(* PLC project Generated.project, CODESYS CODESYS V3.5 SP19 Patch 1 *)
(* stored: creationDateTime 2026-09-19T18:18:07.257453, modificationDateTime 2026-09-19T18:18:07.257453 *)

(* ═══════════════════════════════════════════════════════════════ 🧩 ST_fbWinchCmdArbitration_Context — Contexte de gating treuil (partagé M1/M2) ─────────────────────────────────────────────────────────────── 🎯 Rôle : Encapsuler les faits de gating consommés par FB_WinchCommandArbitrationM1/M2 (benne, synchro, blocage both). Structure UNIQUE partagée par les 2 axes, identifiée par l'instance : M1 ignore le chemin benne, M2 le consomme. 📤 Producteur : PRG_04_Treuils_Benne (câblage). 📄 Doc : DOC/AF/AF_Partie-10_Fonction_Winch_v2.1.md 🔌 Action benne : 2 bits BOOL directionnels M2 issus de FB_Bucket. ═══════════════════════════════════════════════════════════════ *)
TYPE ST_fbWinchCmdArbitration_Context : STRUCT
  BucketBusy : BOOL;  (* --> [STAT] Action benne en cours (instBucket.Lifecycle.Busy) *)
  BucketM2RunRequest : BOOL;  (* --> [CMD] Commande M2 par la benne active *)
  BucketM2ReqAscent : BOOL;  (* --> [CMD] Demande montée M2 issue benne *)
  BucketM2ReqDescend : BOOL;  (* --> [CMD] Demande descente M2 issue benne *)
  BucketAutoCloseActive : BOOL;  (* --> [STAT] AX10 fermeture auto active (plafond AX10 M2, issu de CtrlAscentMaxStep) *)
  BucketHandoffP1Active : BOOL;  (* --> [STAT] AX10B : fermeture atteinte, M2 maintenu au palier 1 avant transfert couple *)
  WinchBothMotionBlockedByBucket : BOOL;  (* --> [STAT] Mouvement both bloqué par benne (ex CoupledMotionBlockedByBucket) *)
  SyncBlocksAscent : BOOL;  (* --> [STAT] Synchro bloque la montée (SyncMinorDeviationBlocksUp) *)
  SyncBlocksDescent : BOOL;  (* --> [STAT] Synchro bloque la descente (SyncMinorDeviationBlocksDown) *)
  M1AscentAllowed : BOOL;  (* === 🔗 ATOMICITÉ DE LA COMMANDE BOTH : permis agrégés consommés === PRG_04 calcule BothAscentPermit/BothDescendPermit = AND des 4 permits effectifs. En commande both, la commande ne consomme QUE ces agrégats (jamais les permits individuels directement) : les 2 treuils partent ensemble ou aucun (NC-100). --> [SAFE] Fait EffectivePermitM1_Ascent *)
  M1DescendAllowed : BOOL;  (* --> [SAFE] Fait EffectivePermitM1_Descend *)
  M2AscentAllowed : BOOL;  (* --> [SAFE] Fait EffectivePermitM2_Ascent *)
  M2DescendAllowed : BOOL;  (* --> [SAFE] Fait EffectivePermitM2_Descend *)
  BothBlock : BOOL;  (* --> [STAT] Commande Both bloquée (aucun départ possible — diagnostic IHM) *)
END_STRUCT;
END_TYPE
